INTERFACE I_SwivelMovement

PROPERTY P_Return : REFERENCE to ST_CommandReturn
GET
END_GET
END_PROPERTY

METHOD StartMovement
VAR_INPUT
	NumCycles		: UINT;
	Velo			: LREAL;
END_VAR
END_METHOD

END_INTERFACE

(* stored: Version 1.1.0.1
   Itf I_SwivelMovement: Id {0348cc1a-8e52-4042-b348-bde316debd0b}
   Property P_Return: Id {b390e548-9456-494e-b0b1-f20dfb920fb2}
   Get Get: Id {1c14d077-8833-4af0-9d58-469e61364fd8}
   Method StartMovement: Id {391f8881-769c-4447-a6ea-0d644f348673} *)
